// TIA Portal V17 export
// export: Created 2022-07-28T18:03:18.010792Z, ExportSetting None, DisplayName Totally Integrated Automation Portal, DisplayVersion V17, DisplayName TIA Portal Openness, DisplayVersion V17, DisplayName TIA Portal Teamcenter Gateway, DisplayVersion V17, DisplayName TIA Portal Version Control Interface, DisplayVersion V17, DisplayName TIA Portal Test Suite Advanced, DisplayVersion V17, DisplayName SINAMICS Startdrive Advanced, DisplayVersion V17, DisplayName SINAMICS DCC, DisplayVersion V17, DisplayName SINAMICS Startdrive G130, G150, S120, S150, SINAMICS MV, S210, DisplayVersion V17, DisplayName SINAMICS Startdrive G110M, G120, G120C, G120D, G120P, G115D, DisplayVersion V17, DisplayName STEP 7 Professional, DisplayVersion V17, DisplayName SIMATIC Energy Suite, DisplayVersion V17, DisplayName STEP 7 CFC, DisplayVersion V17, DisplayName STEP 7 Safety, DisplayVersion V17, DisplayName WinCC Advanced / Unified PC, DisplayVersion V17, DisplayName SIMATIC Visualization Architect, DisplayVersion V17
TYPE "_MotoHours_Unit"
   STRUCT
      di_SetMotoHours { S7_SetPoint := 'True'} : DInt;   // Set motohours, sec
      di_ActLeftMotoHours { ExternalWritable := 'False'; S7_SetPoint := 'True'} : DInt;   // Actual left motohours to next TC, sec
      di_ActMotoHours { ExternalWritable := 'False'; S7_SetPoint := 'True'} : DInt;   // Actual counter of Motohourses, sec
   END_STRUCT;
END_TYPE
